FUNCTION_BLOCK FB_CalcFocalLengthSingleLens_Test EXTENDS FB_TestSuite
VAR
    nTestID : INT;
END_VAR


nTestID := 0;

TestInvalidDeltaExpectError0FocalLength();

Test0DeltaExpectError0FocalLength();

Test0RadiusExpectError0FocalLength();

// Expected results taken from pcdscalc/be_lens_calcs.py.
// Element = Be. Test Count = 1.
TestValidInputsExpectNoErrorAccurateFocalLength(
    fDelta := 0.005621922785393444,
    fRadius := 0.0001,
    fExpected := 0.008893754309452119
);

// Expected results taken from pcdscalc/be_lens_calcs.py.
// Element = Be. Test Count = 2.
TestValidInputsExpectNoErrorAccurateFocalLength(
    fDelta := 0.005621922785393444,
    fRadius := 0.0051,
    fExpected := 0.45358146978205804
);

// Expected results taken from pcdscalc/be_lens_calcs.py.
// Element = Be. Test Count = 3.
TestValidInputsExpectNoErrorAccurateFocalLength(
    fDelta := 1.7147402940032417e-06,
    fRadius := 0.0001,
    fExpected := 29.15893454819898
);

// Expected results taken from pcdscalc/be_lens_calcs.py.
// Element = Be. Test Count = 4.
TestValidInputsExpectNoErrorAccurateFocalLength(
    fDelta := 1.7147402940032417e-06,
    fRadius := 0.0051,
    fExpected := 1487.105661958148
);

// Expected results taken from pcdscalc/be_lens_calcs.py.
// Element = Be. Test Count = 5.
TestValidInputsExpectNoErrorAccurateFocalLength(
    fDelta := 4.316182378185529e-07,
    fRadius := 0.0001,
    fExpected := 115.84311231310711
);

// Expected results taken from pcdscalc/be_lens_calcs.py.
// Element = Be. Test Count = 6.
TestValidInputsExpectNoErrorAccurateFocalLength(
    fDelta := 4.316182378185529e-07,
    fRadius := 0.0051,
    fExpected := 5907.998727968463
);


METHOD PRIVATE SetInitialDeltaAndRadiusValues
VAR_IN_OUT
    fbCalcXRayDeltaMock : FB_CalcXRayDeltaMock;
END_VAR

fbCalcXRayDeltaMock.SetValid();
END_METHOD


METHOD PRIVATE Test0DeltaExpectError0FocalLength
VAR
    fbCalcXRayDeltaMock : FB_CalcXRayDeltaMock;
    // Subject under test
    fbCalcFocalLengthSingleLens : FB_CalcFocalLengthSingleLens(iCalcXRayDelta := fbCalcXRayDeltaMock);
    fResult : LREAL;
END_VAR

TEST('Test0DeltaExpectError0FocalLength');

// Test Fixture
SetInitialDeltaAndRadiusValues(fbCalcXRayDeltaMock := fbCalcXRayDeltaMock);

fbCalcXRayDeltaMock.SetResult(0.0);

fResult := fbCalcFocalLengthSingleLens.Calculate(
    sElementName := 'Be',
    fRadius := 1.0
);

AssertTrue(
    Condition := fbCalcFocalLengthSingleLens.GetError(),
    Message := 'Expected bError bit to be true but it was false.'
);

AssertTrue(
    Condition := fbCalcFocalLengthSingleLens.GetErrorMsg() <> '',
    Message := 'Expected sErrorMsg to not be empty.'
);

AssertEquals_LREAL(
    Expected := 0,
    Actual := fResult,
    Delta := 0,
    Message := 'Calculated focal length should be 0 when an error is detected.'
);

TEST_FINISHED();
END_METHOD


METHOD PRIVATE Test0RadiusExpectError0FocalLength
VAR
    fbCalcXRayDeltaMock : FB_CalcXRayDeltaMock;
    // Subject under test
    fbCalcFocalLengthSingleLens : FB_CalcFocalLengthSingleLens(iCalcXRayDelta := fbCalcXRayDeltaMock);
    fResult : LREAL;
END_VAR

TEST('Test0RadiusExpectError0FocalLength');

// Test Fixture
SetInitialDeltaAndRadiusValues(fbCalcXRayDeltaMock := fbCalcXRayDeltaMock);


fResult := fbCalcFocalLengthSingleLens.Calculate(
    sElementName := 'Be',
    fRadius := 0.0
);

AssertTrue(
    Condition := fbCalcFocalLengthSingleLens.GetError(),
    Message := 'Expected bError bit to be true but it was false.'
);

AssertTrue(
    Condition := fbCalcFocalLengthSingleLens.GetErrorMsg() <> '',
    Message := 'Expected sErrorMsg to not be empty.'
);

AssertEquals_LREAL(
    Expected := 0,
    Actual := fResult,
    Delta := 0,
    Message := 'Calculated focal length should be 0 when an error is detected.'
);

TEST_FINISHED();
END_METHOD


METHOD PRIVATE TestInvalidDeltaExpectError0FocalLength
VAR
    fbCalcXRayDeltaMock : FB_CalcXRayDeltaMock;
    // Subject under test
    fbCalcFocalLengthSingleLens : FB_CalcFocalLengthSingleLens(iCalcXRayDelta := fbCalcXRayDeltaMock);
    fResult : LREAL;
END_VAR

TEST('TestInvalidDeltaExpectError0FocalLength');

// Test fixture
SetInitialDeltaAndRadiusValues(fbCalcXRayDeltaMock := fbCalcXRayDeltaMock);

fbCalcXRayDeltaMock.SetError(sMsg := 'Error');

fResult := fbCalcFocalLengthSingleLens.Calculate(
    sElementName := 'Be',
    fRadius := 1.0
);

AssertTrue(
    Condition := fbCalcFocalLengthSingleLens.GetError(),
    Message := 'Expected bError bit to be true but it was false.'
);

AssertTrue(
    Condition := fbCalcFocalLengthSingleLens.GetErrorMsg() <> '',
    Message := 'Expected sErrorMsg to not be empty.'
);

AssertEquals_LREAL(
    Expected := 0,
    Actual := fResult,
    Delta := 0,
    Message := 'Calculated focal length should be 0 when an error is detected.'
);

TEST_FINISHED();
END_METHOD


METHOD PRIVATE TestValidInputsExpectNoErrorAccurateFocalLength
VAR_INPUT
    fDelta : LREAL;
    fRadius : LREAL;

    fExpected : LREAL;
END_VAR
VAR
    fbCalcXRayDeltaMock : FB_CalcXRayDeltaMock;
    // Subject under test
    fbCalcFocalLengthSingleLens : FB_CalcFocalLengthSingleLens(iCalcXRayDelta := fbCalcXRayDeltaMock);
    fResult : LREAL;
END_VAR

TEST(CONCAT(STR1 := 'TestValidInputsExpectNoErrorAccurateFocalLength ID: ',
            STR2 := INT_TO_STRING(nTestID)));

// Test fixture
SetInitialDeltaAndRadiusValues(fbCalcXRayDeltaMock := fbCalcXRayDeltaMock);

fbCalcXRayDeltaMock.SetResult(fDelta);

// Here the test starts

fResult := fbCalcFocalLengthSingleLens.Calculate(
    sElementName := 'Be',
    fRadius := fRadius
);

AssertFalse(
    Condition := fbCalcFocalLengthSingleLens.GetError(),
    Message := 'Expected bError bit to be false but it was true.'
);

AssertFalse(
    Condition := fbCalcFocalLengthSingleLens.GetErrorMsg() <> '',
    Message := 'Expected sErrorMsg to be empty.'
);

AssertEquals_LREAL(
    Expected := fExpected,
    Actual := fResult,
    Delta := ABS(0.001 * fExpected),
    Message := 'Calculated focal length did not calculate close enough to the expected value.'
);

TEST_FINISHED();

nTestID := nTestID + 1;
END_METHOD

END_FUNCTION_BLOCK

(* stored: Version 1.1.0.1
   POU FB_CalcFocalLengthSingleLens_Test: Id {85175de0-d809-48a0-9035-d5cabefef591}, SpecialFunc None
   Method SetInitialDeltaAndRadiusValues: Id {bdf9ec0b-14ec-48c2-a21f-eb2530271dd3}
   Method Test0DeltaExpectError0FocalLength: Id {884decc0-7ccd-43be-b539-b042f489f0ce}
   Method Test0RadiusExpectError0FocalLength: Id {2678e1cc-84be-4dd6-bdd3-4144cce0f4be}
   Method TestInvalidDeltaExpectError0FocalLength: Id {8ce1ae93-c963-4cfd-a51e-bb3ddb1a3cf0}
   Method TestValidInputsExpectNoErrorAccurateFocalLength: Id {ecdb3377-455a-469a-8223-4fdf93173dff} *)
